PROGRAM SmokeControl
VAR
	StartupDone: BOOL;
	GreenMasterSmokeControl: GreenMasterSmokeControl; 
	Parameters: reference to GreenMasterBaseParameters;
END_VAR

IF NOT StartupDone THEN
	Parameters REF= Main.GreenMaster.GetParameters();
	StartupDone := TRUE;
END_IF

GreenMasterSmokeControl(EN := TRUE, Parameters := Parameters, ParametersSC := Main.GreenMaster.GetParametersSC());

END_PROGRAM

(* stored: Version 1.1.0.1, ProductVersion 3.1.4024.6
   POU SmokeControl: Id {ece165da-f1ed-4d49-8ac5-2cb738a1f4d6}, SpecialFunc None *)
